{attribute 'GeneratedUsingTerminal: EK1122-0000-0018'}
{attribute addProperty BoxType "EK1122-0000-0018"}
{attribute addProperty Id "Beckhoff_EJ2xxxsub_EK1100EK1100_AB5A94672"}
{attribute addProperty CRC "3176198815"}
{attribute addProperty Size "2"}
TYPE Beckhoff_EJ2xxxEK1122_BD50F29F EXTENDS EK1122_AB5A9467 :
STRUCT
	{attribute addProperty Name "Beckhoff_EJ2xxxsub_EK1100"}
	Beckhoff_EJ2xxxsub_EK1100 : EK1100_AB5A9467;
END_STRUCT
END_TYPE

(* stored: Version 1.2.0.0, ProductVersion 3.1.4024.9
   DUT Beckhoff_EJ2xxxEK1122_BD50F29F: Id {e0d41630-8dda-4cb3-a9b4-4e5162f2ba36} *)
